(* CoDeSys 2.3.9.41 project: telejka0.pro *)
(* Libraries: Standard.lib 4.10.05 11:14:46, IecSfc.lib 13.4.06 15:51:28, SYSLIBCALLBACK.LIB 26.9.08 16:43:52 *)

(* Global variable list: Global_Variables *)
VAR_GLOBAL
	observer: BOOL;
	Warning: BOOL;
	Stop: BOOL;
END_VAR

(* POU PLC_PRG, FBD *)
PROGRAM PLC_PRG
VAR
	Trig1: R_TRIG;
	Trig2: F_TRIG;
	Timer1: TOF;

	Timer2: TON;

END_VAR
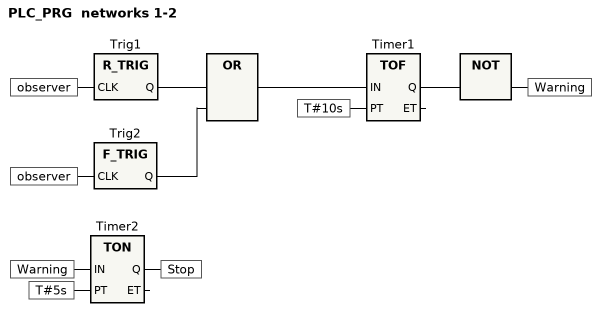
_FBD_ (* Function Block Diagram *)
NETWORK 1
	NOT Timer1:TOF(IN: OR(Trig1:R_TRIG(CLK: observer), Trig2:F_TRIG(CLK: observer)), PT: T#10s) => Warning
NETWORK 2
	Timer2:TON(IN: Warning, PT: T#5s) => Stop
_END_FBD_
(* the same logic as Structured Text *)
(* Network 1 *)
Trig1(CLK := observer);
Trig2(CLK := observer);
Timer1(IN := Trig1.Q OR Trig2.Q, PT := T#10s);
Warning := NOT Timer1.Q;
(* Network 2 *)
Timer2(IN := Warning, PT := T#5s);
Stop := Timer2.Q;
END_PROGRAM

(* POU Machine, SFC *)
PROGRAM Machine
VAR
END_VAR
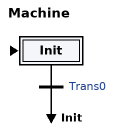
INITIAL_STEP Init:
END_STEP
TRANSITION FROM Init TO Init := Trans0;
END_TRANSITION
END_PROGRAM
